FUNCTION_BLOCK GritScreenBasic (* Basic Function Block Type *)
  (* Standard: 61499-2 *)
  (* Version 0.0, 6/16/2026, Schneider Electric, Template *)
  PACKAGE SE.Nereda;
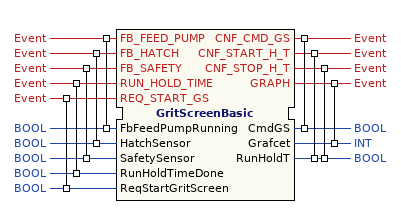
  EVENT_INPUT
    FB_FEED_PUMP WITH FbFeedPumpRunning;
    FB_HATCH WITH HatchSensor;
    FB_SAFETY WITH SafetySensor;
    RUN_HOLD_TIME WITH RunHoldTimeDone;
    REQ_START_GS WITH ReqStartGritScreen;
  END_EVENT
  EVENT_OUTPUT
    CNF_CMD_GS WITH CmdGS;
    CNF_START_H_T WITH RunHoldT;
    CNF_STOP_H_T WITH RunHoldT;
    GRAPH WITH Grafcet;
  END_EVENT
  VAR_INPUT
    FbFeedPumpRunning : BOOL;
    HatchSensor : BOOL;
    SafetySensor : BOOL;
    RunHoldTimeDone : BOOL;
    ReqStartGritScreen : BOOL;
  END_VAR
  VAR_OUTPUT
    CmdGS : BOOL;
    Grafcet : INT;
    RunHoldT : BOOL;
  END_VAR
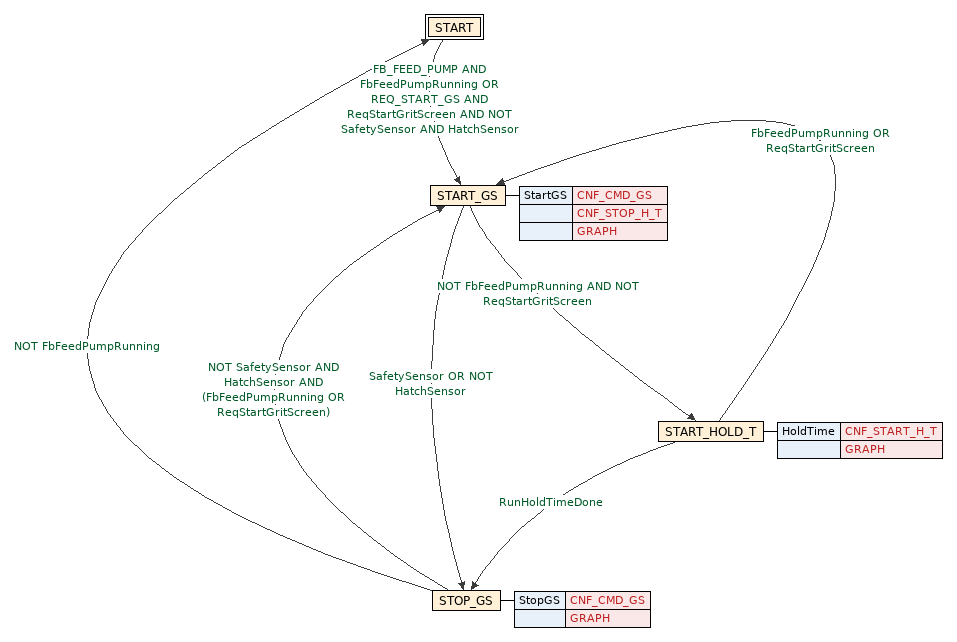
  EC_STATES
    START; (* Initial State *)
    START_GS : StartGS -> CNF_CMD_GS, -> CNF_STOP_H_T, -> GRAPH;
    STOP_GS : StopGS -> CNF_CMD_GS, -> GRAPH;
    START_HOLD_T : HoldTime -> CNF_START_H_T, -> GRAPH;
  END_STATES
  EC_TRANSITIONS
    START TO START_GS := FB_FEED_PUMP AND FbFeedPumpRunning OR REQ_START_GS AND ReqStartGritScreen AND NOT SafetySensor AND HatchSensor;
    START_GS TO START_HOLD_T := NOT FbFeedPumpRunning AND NOT ReqStartGritScreen;
    START_HOLD_T TO STOP_GS := RunHoldTimeDone;
    START_GS TO STOP_GS := SafetySensor OR NOT HatchSensor;
    STOP_GS TO START_GS := NOT SafetySensor AND HatchSensor AND (FbFeedPumpRunning OR ReqStartGritScreen);
    STOP_GS TO START := NOT FbFeedPumpRunning;
    START_HOLD_T TO START_GS := FbFeedPumpRunning OR ReqStartGritScreen;
  END_TRANSITIONS
  ALGORITHM StartGS IN ST:
;
Grafcet := 1;
CmdGS := TRUE;
RunHoldT := FALSE;
  END_ALGORITHM
  ALGORITHM HoldTime IN ST:
;
Grafcet := 3;
RunHoldT := TRUE;
  END_ALGORITHM
  ALGORITHM StopGS IN ST:
;
Grafcet := 2;
CmdGS := FALSE;
RunHoldT := FALSE;
  END_ALGORITHM
END_FUNCTION_BLOCK
